# EPICS autosave request: pokaApp/Db/DCMotorServer.req
$(P)ramp_time
$(P)v_top
$(P)v_base
$(P)m1.DESC
$(P)m1:step:size
$(P)m1:step:change.C
$(P)m1:step:change.D
$(P)m2.DESC
$(P)m2:step:size
$(P)m2:step:change.C
$(P)m2:step:change.D
$(P)m3.DESC
$(P)m3:step:size
$(P)m3:step:change.C
$(P)m3:step:change.D
$(P)m4.DESC
$(P)m4:step:size
$(P)m4:step:change.C
$(P)m4:step:change.D
